FUNCTION_BLOCK ButtonManager
VAR_INPUT
END_VAR
VAR_OUTPUT
END_VAR
VAR
	DI_StartButton_Terminal1 AT%I*: BOOL;
	DI_StartButton_Terminal2 AT%I*: BOOL;	
	DI_StartButton_Terminal3 AT%I*: BOOL;	
	DI_StartButton_Door AT%I*: BOOL;	
	DI_StartButton_LightBarrier AT%I*: BOOL;	
	
	DI_StopButton_Door AT%I*: BOOL;	
	DI_StopButton_LightBarrier AT%I*: BOOL;	
	
	DI_EStopButton_Terminal1 AT%I*: BOOL;
	DI_EStopButton_Terminal2 AT%I*: BOOL;	
	DI_EStopButton_Terminal3 AT%I*: BOOL;	
	//DI_EStopButton_Door AT%I*: BOOL;     //currently not connected to PLC
	DI_EStopButton_LightBarrier AT%I*: BOOL;
	
	DI_ResetButton_Door AT%I*: BOOL;
	DI_ResetButton_LightBarrier AT%I*: BOOL;
END_VAR

//manages the Start-, Stop-, Reset- and EStop-Buttons

PROPERTY EStop : BOOL
GET
// EStops physically implemented as Failsafe, they return True, when not pressed.
//for better handling this is reversed here
EStop := NOT DI_EStopButton_LightBarrier OR NOT DI_EStopButton_Terminal1 OR NOT DI_EStopButton_Terminal2 OR NOT DI_EStopButton_Terminal3;
END_GET
END_PROPERTY

PROPERTY Reset : BOOL
GET
Reset := DI_ResetButton_Door OR DI_ResetButton_LightBarrier;
END_GET
END_PROPERTY

PROPERTY Start : BOOL
GET
Start := DI_StartButton_Door OR DI_StartButton_LightBarrier OR DI_StartButton_Terminal1 OR DI_StartButton_Terminal2 OR DI_StartButton_Terminal3;
END_GET
END_PROPERTY

PROPERTY Stop : BOOL
GET
// EStops physically implemented as Failsafe, they return True, when not pressed.
//for better handling this is reversed here
Stop := NOT DI_StopButton_Door OR NOT DI_StopButton_LightBarrier;
END_GET
END_PROPERTY

END_FUNCTION_BLOCK

(* stored: Version 1.1.0.1, ProductVersion 3.1.4024.12
   POU ButtonManager: Id {84af5a22-f6c3-40e7-b04e-7fad7f555d5d}, SpecialFunc None
   Property EStop: Id {f2e58e39-487e-465d-ad45-ba0a8a086814}
   Get Get: Id {2a69571f-d77c-4030-b740-f787e7a2f46e}
   Property Reset: Id {50140a7c-29e4-41f4-8ea5-a56af778457c}
   Get Get: Id {7d9203e3-d9ce-420a-b885-d6567b56d269}
   Property Start: Id {14840054-998c-46d6-a4df-8b4cf544a550}
   Get Get: Id {9f159ac2-3de3-4abc-a995-447a12ca6251}
   Property Stop: Id {1d979780-ca09-4cb7-bd2b-dc7ff7cb8d77}
   Get Get: Id {97c4fa01-0e19-4f4e-b309-812d451e5911} *)
